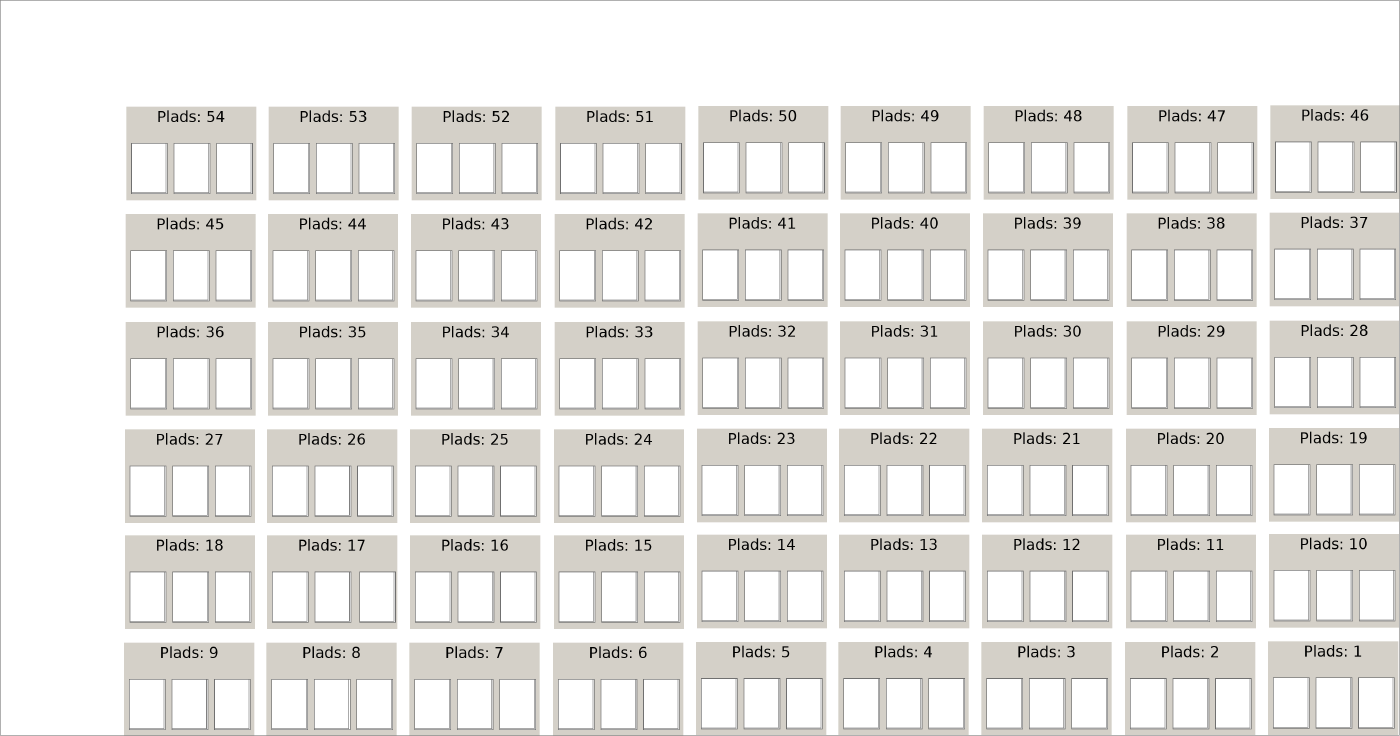
VISUALIZATION Visualization_Pos  // 2007x1056
    Textfield (1818,920 186x134), "Plads: 1", colour toggle: MAIN.Occ
    Button (1886,972 52x73), colour toggle: HMI.Lamp1_Green
        toggle HMI.Lamp1_Green
    Button (1825,972 52x73), colour toggle: HMI.Lamp1_Metal
    Button (1947,972 52x73), colour toggle: HMI.Lamp1_Blue
        toggle HMI.Lamp1_Blue
    Textfield (1613,921 186x134), "Plads: 2", colour toggle: MAIN.Occ
    Button (1681,973 52x73), colour toggle: HMI.Lamp2_Green
    Button (1620,973 52x73)
    Button (1742,973 52x73), colour toggle: HMI.Lamp2_Blue
    Textfield (1407,921 186x134), "Plads: 3", colour toggle: MAIN.Occ
    Button (1475,973 52x73), colour toggle: HMI.Lamp3_Green
    Button (1414,973 52x73), colour toggle: HMI.Lamp3_Metal
    Button (1536,973 52x73), colour toggle: HMI.Lamp3_Blue
    Textfield (1202,921 186x134), "Plads: 4"
    Button (1270,973 52x73), colour toggle: HMI.Lamp4_Green
    Button (1209,973 52x73), colour toggle: HMI.Lamp4_Metal
    Button (1331,973 52x73), colour toggle: HMI.Lamp4_Blue
    Textfield (998,921 186x134), "Plads: 5"
    Button (1066,973 52x73)
    Button (1005,973 52x73)
    Button (1127,973 52x73), colour toggle: MAIN.bStart
    Textfield (793,922 186x134), "Plads: 6"
    Button (861,974 52x73), colour toggle: HMI.Lamp6_Green
    Button (800,974 52x73), colour toggle: HMI.Lamp6_Metal
    Button (922,974 52x73), colour toggle: HMI.Lamp6_Blue
    Textfield (587,922 186x134), "Plads: 7"
    Button (655,974 52x73), colour toggle: HMI.Lamp7_Green
    Button (594,974 52x73), colour toggle: HMI.Lamp7_Metal
    Button (716,974 52x73), colour toggle: HMI.Lamp7_Blue
    Textfield (382,922 186x134), "Plads: 8"
    Button (450,974 52x73), colour toggle: HMI.Lamp8_Green
    Button (389,974 52x73), colour toggle: HMI.Lamp8_Metal
    Button (511,974 52x73), colour toggle: HMI.Lamp8_Blue
    Textfield (178,922 186x134), "Plads: 9"
    Button (246,974 52x73), colour toggle: HMI.Lamp9_Green
    Button (185,974 52x73), colour toggle: HMI.Lamp9_Metal
    Button (307,974 52x73), colour toggle: HMI.Lamp9_Blue
    Textfield (1819,766 186x134), "Plads: 10"
    Button (1887,818 52x73), colour toggle: HMI.Lamp10_Green
    Button (1826,818 52x73), colour toggle: HMI.Lamp10_Metal
    Button (1948,818 52x73), colour toggle: HMI.Lamp10_Blue
    Textfield (1614,767 186x134), "Plads: 11"
    Button (1682,819 52x73), colour toggle: HMI.Lamp11_Green
    Button (1621,819 52x73), colour toggle: HMI.Lamp11_Metal
    Button (1743,819 52x73), colour toggle: HMI.Lamp11_Blue
    Textfield (1408,767 186x134), "Plads: 12"
    Button (1476,819 52x73), colour toggle: HMI.Lamp12_Green
    Button (1415,819 52x73), colour toggle: HMI.Lamp12_Metal
    Button (1537,819 52x73), colour toggle: HMI.Lamp12_Blue
    Textfield (1203,767 186x134), "Plads: 13"
    Button (1271,819 52x73), colour toggle: HMI.Lamp13_Green
    Button (1210,819 52x73), colour toggle: HMI.Lamp13_Metal
    Button (1332,819 52x73), colour toggle: HMI.Lamp13_Blue
    Textfield (999,767 186x134), "Plads: 14"
    Button (1067,819 52x73), colour toggle: HMI.Lamp14_Green
    Button (1006,819 52x73), colour toggle: HMI.Lamp14_Metal
    Button (1128,819 52x73), colour toggle: HMI.Lamp14_Blue
    Textfield (794,768 186x134), "Plads: 15"
    Button (862,820 52x73), colour toggle: HMI.Lamp15_Green
    Button (801,820 52x73), colour toggle: HMI.Lamp15_Metal
    Button (923,820 52x73), colour toggle: HMI.Lamp15_Blue
    Textfield (588,768 186x134), "Plads: 16"
    Button (656,820 52x73), colour toggle: HMI.Lamp16_Green
    Button (595,820 52x73), colour toggle: HMI.Lamp16_Metal
    Button (717,820 52x73), colour toggle: HMI.Lamp16_Blue
    Textfield (383,768 186x134), "Plads: 17"
    Button (451,820 52x73), colour toggle: HMI.Lamp17_Green
    Button (390,820 52x73), colour toggle: HMI.Lamp17_Metal
    Button (515,820 52x73), colour toggle: HMI.Lamp17_Blue
    Textfield (179,768 186x134), "Plads: 18"
    Button (247,820 52x73), colour toggle: HMI.Lamp18_Green
    Button (186,820 52x73), colour toggle: HMI.Lamp18_Metal
    Button (308,820 52x73), colour toggle: HMI.Lamp18_Blue
    Textfield (1819,614 186x134), "Plads: 19"
    Button (1887,666 52x73), colour toggle: HMI.Lamp19_Green
    Button (1826,666 52x73), colour toggle: HMI.Lamp19_Metal
    Button (1948,666 52x73), colour toggle: HMI.Lamp19_Blue
    Textfield (1614,615 186x134), "Plads: 20"
    Button (1682,667 52x73), colour toggle: HMI.Lamp20_Green
    Button (1621,667 52x73), colour toggle: HMI.Lamp20_Metal
    Button (1743,667 52x73), colour toggle: HMI.Lamp20_Blue
    Textfield (1408,615 186x134), "Plads: 21"
    Button (1476,667 52x73), colour toggle: HMI.Lamp21_Green
    Button (1415,667 52x73), colour toggle: HMI.Lamp21_Metal
    Button (1537,667 52x73), colour toggle: HMI.Lamp21_Blue
    Textfield (1203,615 186x134), "Plads: 22"
    Button (1271,667 52x73), colour toggle: HMI.Lamp22_Green
    Button (1210,667 52x73), colour toggle: HMI.Lamp22_Metal
    Button (1332,667 52x73), colour toggle: HMI.Lamp22_Blue
    Textfield (999,615 186x134), "Plads: 23"
    Button (1067,667 52x73), colour toggle: HMI.Lamp23_Green
    Button (1006,667 52x73), colour toggle: HMI.Lamp23_Metal
    Button (1128,667 52x73), colour toggle: HMI.Lamp23_Blue
    Textfield (794,616 186x134), "Plads: 24"
    Button (862,668 52x73), colour toggle: HMI.Lamp24_Green
    Button (801,668 52x73), colour toggle: HMI.Lamp24_Metal
    Button (923,668 52x73), colour toggle: HMI.Lamp24_Blue
    Textfield (588,616 186x134), "Plads: 25"
    Button (656,668 52x73), colour toggle: HMI.Lamp25_Green
    Button (595,668 52x73), colour toggle: HMI.Lamp25_Metal
    Button (717,668 52x73), colour toggle: HMI.Lamp25_Blue
    Textfield (383,616 186x134), "Plads: 26"
    Button (451,668 52x73), colour toggle: HMI.Lamp26_Green
    Button (390,668 52x73), colour toggle: HMI.Lamp26_Metal
    Button (512,668 52x73), colour toggle: HMI.Lamp26_Blue
    Textfield (179,616 186x134), "Plads: 27"
    Button (247,668 52x73), colour toggle: HMI.Lamp27_Green
    Button (186,668 52x73), colour toggle: HMI.Lamp27_Metal
    Button (308,668 52x73), colour toggle: HMI.Lamp27_Blue
    Textfield (1820,460 186x134), "Plads: 28"
    Button (1888,512 52x73), colour toggle: HMI.Lamp28_Green
    Button (1827,512 52x73), colour toggle: HMI.Lamp28_Metal
    Button (1949,512 52x73), colour toggle: HMI.Lamp28_Blue
    Textfield (1615,461 186x134), "Plads: 29"
    Button (1683,513 52x73), colour toggle: HMI.Lamp29_Green
    Button (1622,513 52x73), colour toggle: HMI.Lamp29_Metal
    Button (1744,513 52x73), colour toggle: HMI.Lamp29_Blue
    Textfield (1409,461 186x134), "Plads: 30"
    Button (1477,513 52x73), colour toggle: HMI.Lamp30_Green
    Button (1416,513 52x73), colour toggle: HMI.Lamp30_Metal
    Button (1538,513 52x73), colour toggle: HMI.Lamp30_Blue
    Textfield (1204,461 186x134), "Plads: 31"
    Button (1272,513 52x73), colour toggle: HMI.Lamp31_Green
    Button (1211,513 52x73), colour toggle: HMI.Lamp31_Metal
    Button (1333,513 52x73), colour toggle: HMI.Lamp31_Blue
    Textfield (1000,461 186x134), "Plads: 32"
    Button (1068,513 52x73), colour toggle: HMI.Lamp32_Green
    Button (1007,513 52x73), colour toggle: HMI.Lamp32_Metal
    Button (1129,513 52x73), colour toggle: HMI.Lamp32_Blue
    Textfield (795,462 186x134), "Plads: 33"
    Button (863,514 52x73), colour toggle: HMI.Lamp33_Green
    Button (802,514 52x73), colour toggle: HMI.Lamp33_Metal
    Button (924,514 52x73), colour toggle: HMI.Lamp33_Blue
    Textfield (589,462 186x134), "Plads: 34"
    Button (657,514 52x73), colour toggle: HMI.Lamp34_Blue
    Button (596,514 52x73), colour toggle: HMI.Lamp34_Metal
    Button (718,514 52x73), colour toggle: HMI.Lamp34_Blue
    Textfield (384,462 186x134), "Plads: 35"
    Button (452,514 52x73), colour toggle: HMI.Lamp35_Green
    Button (391,514 52x73), colour toggle: HMI.Lamp35_Metal
    Button (513,514 52x73), colour toggle: HMI.Lamp35_Blue
    Textfield (180,462 186x134), "Plads: 36"
    Button (248,514 52x73), colour toggle: HMI.Lamp36_Green
    Button (187,514 52x73), colour toggle: HMI.Lamp36_Metal
    Button (309,514 52x73), colour toggle: HMI.Lamp36_Blue
    Textfield (1820,305 186x134), "Plads: 37"
    Button (1888,357 52x73), colour toggle: HMI.Lamp37_Green
    Button (1827,357 52x73), colour toggle: HMI.Lamp37_Metal
    Button (1949,357 52x73), colour toggle: HMI.Lamp37_Blue
    Textfield (1615,306 186x134), "Plads: 38"
    Button (1683,358 52x73), colour toggle: HMI.Lamp38_Green
    Button (1622,358 52x73), colour toggle: HMI.Lamp38_Metal
    Button (1744,358 52x73), colour toggle: HMI.Lamp38_Blue
    Textfield (1409,306 186x134), "Plads: 39"
    Button (1477,358 52x73), colour toggle: HMI.Lamp39_Green
    Button (1416,358 52x73), colour toggle: HMI.Lamp39_Metal
    Button (1538,358 52x73), colour toggle: HMI.Lamp39_Blue
    Textfield (1204,306 186x134), "Plads: 40"
    Button (1272,358 52x73), colour toggle: HMI.Lamp40_Green
    Button (1211,358 52x73), colour toggle: HMI.Lamp40_Metal
    Button (1333,358 52x73), colour toggle: HMI.Lamp40_Blue
    Textfield (1000,306 186x134), "Plads: 41"
    Button (1068,358 52x73), colour toggle: HMI.Lamp41_Green
    Button (1007,358 52x73), colour toggle: HMI.Lamp41_Metal
    Button (1129,358 52x73), colour toggle: HMI.Lamp41_Blue
    Textfield (795,307 186x134), "Plads: 42"
    Button (863,359 52x73), colour toggle: HMI.Lamp42_Green
    Button (802,359 52x73), colour toggle: HMI.Lamp42_Metal
    Button (924,359 52x73), colour toggle: HMI.Lamp42_Blue
    Textfield (589,307 186x134), "Plads: 43"
    Button (657,359 52x73), colour toggle: HMI.Lamp43_Green
    Button (596,359 52x73), colour toggle: HMI.Lamp43_Metal
    Button (718,359 52x73), colour toggle: HMI.Lamp43_Blue
    Textfield (384,307 186x134), "Plads: 44"
    Button (452,359 52x73), colour toggle: HMI.Lamp44_Green
    Button (391,359 52x73), colour toggle: HMI.Lamp44_Metal
    Button (513,359 52x73), colour toggle: HMI.Lamp44_Blue
    Textfield (180,307 186x134), "Plads: 45"
    Button (248,359 52x73), colour toggle: HMI.Lamp45_Green
    Button (187,359 52x73), colour toggle: HMI.Lamp45_Metal
    Button (309,359 52x73), colour toggle: HMI.Lamp45_Blue
    Textfield (1821,151 186x134), "Plads: 46"
    Button (1889,203 52x73), colour toggle: HMI.Lamp46_Green
    Button (1828,203 52x73), colour toggle: HMI.Lamp46_Metal
    Button (1950,203 52x73), colour toggle: HMI.Lamp46_Blue
    Textfield (1616,152 186x134), "Plads: 47"
    Button (1684,204 52x73), colour toggle: HMI.Lamp47_Green
    Button (1623,204 52x73), colour toggle: HMI.Lamp47_Metal
    Button (1745,204 52x73), colour toggle: HMI.Lamp47_Blue
    Textfield (1410,152 186x134), "Plads: 48"
    Button (1478,204 52x73), colour toggle: HMI.Lamp48_Green
    Button (1417,204 52x73), colour toggle: HMI.Lamp48_Metal
    Button (1539,204 52x73), colour toggle: HMI.Lamp48_Blue
    Textfield (1205,152 186x134), "Plads: 49"
    Button (1273,204 52x73), colour toggle: HMI.Lamp49_Green
    Button (1212,204 52x73), colour toggle: HMI.Lamp49_Metal
    Button (1334,204 52x73), colour toggle: HMI.Lamp49_Blue
    Textfield (1001,152 186x134), "Plads: 50"
    Button (1069,204 52x73), colour toggle: HMI.Lamp50_Green
    Button (1008,204 52x73), colour toggle: HMI.Lamp50_Metal
    Button (1130,204 52x73), colour toggle: HMI.Lamp50_Blue
    Textfield (796,153 186x134), "Plads: 51"
    Button (864,205 52x73), colour toggle: HMI.Lamp51_Green
    Button (803,205 52x73), colour toggle: HMI.Lamp51_Metal
    Button (925,205 52x73), colour toggle: HMI.Lamp51_Blue
    Textfield (590,153 186x134), "Plads: 52"
    Button (658,205 52x73), colour toggle: HMI.Lamp52_Green
    Button (597,205 52x73), colour toggle: HMI.Lamp52_Metal
    Button (719,205 52x73), colour toggle: HMI.Lamp52_Blue
    Textfield (385,153 186x134), "Plads: 53"
    Button (453,205 52x73), colour toggle: HMI.Lamp53_Green
    Button (392,205 52x73), colour toggle: HMI.Lamp53_Metal
    Button (514,205 52x73), colour toggle: HMI.Lamp53_Blue
    Textfield (181,153 186x134), "Plads: 54"
    Button (249,205 52x73), colour toggle: HMI.Lamp54_Green
    Button (188,205 52x73), colour toggle: HMI.Lamp54_Metal
    Button (310,205 52x73), colour toggle: HMI.Lamp54_Blue
END_VISUALIZATION

(* stored: Version 1.1.0.1, ProductVersion 3.1.4024.3
   Visu Visualization_Pos: Id {9d639068-d133-4714-9808-b62686035d6a} *)
